DATA_BLOCK "Cyclic Input Data"
{ S7_Optimized_Access := 'FALSE' }
VERSION : 0.1
NON_RETAIN
   STRUCT
      Static_1 : "Measuring Block Read";
   END_STRUCT;


BEGIN

END_DATA_BLOCK

